// TwinCAT 3 PLC project PLC1
// ProgramVersion: 3.1.4022.7
// libraries:
//   Tc2_Standard, * (Beckhoff Automation GmbH)
//   Tc2_System, * (Beckhoff Automation GmbH)
//   Tc3_Module, * (Beckhoff Automation GmbH)
// project tree:
//   FBs/ FB_Publisher.TcPOU, FB_Subscriber.TcPOU
//   ITFs/ I_Publisher.TcIO, I_Subscriber.TcIO
//   / Param.TcGVL, PlcTask.TcTTO
//   POUs/ MAIN.TcPOU
// real-time tasks:
//   TASK PlcTask: cycle T#10ms, priority 20, ADS port 350

CONFIGURATION PLC1
    RESOURCE PLC ON TwinCAT3
        TASK PlcTask(INTERVAL := T#10ms, PRIORITY := 20);
        PROGRAM MAIN WITH PlcTask : MAIN;
    END_RESOURCE
END_CONFIGURATION

// ---- Param.TcGVL
{attribute 'qualified_only'}
VAR_GLOBAL CONSTANT
	MaxSubscribers : INT := 5;
END_VAR

// ---- ITFs/I_Publisher.TcIO
INTERFACE I_Publisher

METHOD AddSubscriber : BOOL
VAR_INPUT
	ipSubscriber : I_Subscriber;
END_VAR
END_METHOD

METHOD RemoveSubscriber : BOOL
VAR_INPUT
	ipSubscriber : I_Subscriber;
END_VAR
END_METHOD

END_INTERFACE

// ---- ITFs/I_Subscriber.TcIO
INTERFACE I_Subscriber

METHOD Update : BOOL
VAR_INPUT
	Value : LREAL;
END_VAR
END_METHOD

END_INTERFACE

// ---- POUs/MAIN.TcPOU
PROGRAM MAIN
VAR
	(*Design Pattern Blocks *)
	fbPublisher 	: FB_Publisher;
	fbSubscriber 	: ARRAY[1..Param.MaxSubscribers] OF FB_Subscriber;
	
	(* UI Values *)
	AddSub			: ARRAY[1..Param.MaxSubscribers] OF BOOL;
	DeleteSub		: ARRAY[1..Param.MaxSubscribers] OF BOOL;
	i				: INT;
END_VAR

fbPublisher();

FOR i := 1 TO Param.MaxSubscribers DO
	
	IF (AddSub[i]) THEN
		fbPublisher.AddSubscriber(fbSubscriber[i]);
		AddSub[i] := FALSE;
	END_IF

	IF (DeleteSub[i]) THEN
		fbPublisher.RemoveSubscriber(fbSubscriber[i]);
		DeleteSub[i] := FALSE;
	END_IF
	
END_FOR

END_PROGRAM

// ---- FBs/FB_Publisher.TcPOU
FUNCTION_BLOCK PUBLIC FB_Publisher IMPLEMENTS I_Publisher
VAR	
	fbDelay				: TON;
	fbDrand				: DRAND;
	_Value				: LREAL;
	aSubscribers		: ARRAY [1..Param.MaxSubscribers] OF I_Subscriber;
END_VAR

// creates every sec a random value and invoke the update method
fbDelay(IN := TRUE, PT := T#1S);
IF (fbDelay.Q) THEN	
	fbDelay(IN := FALSE);	
	fbDrand(SEED := 0);
	_Value := fbDrand.Num * 1234.5;
	NotifySubscribers();
END_IF

PROPERTY ActualValue : LREAL
GET
ActualValue := THIS^._Value;
END_GET
END_PROPERTY

METHOD PUBLIC AddSubscriber : BOOL
VAR_INPUT
	ipSubscriber	: I_Subscriber;
END_VAR
VAR
	nIndex					: INT := 0;
END_VAR
AddSubscriber := FALSE;
IF (ipSubscriber = 0) THEN
	RETURN;
END_IF

// is the observer already registered?
FOR nIndex := 1 TO Param.MaxSubscribers DO	
	IF (THIS^.aSubscribers[nIndex] = ipSubscriber) THEN
		RETURN;
	END_IF
END_FOR

// save the observer object into the array of observers and send the actual value
FOR nIndex := 1 TO Param.MaxSubscribers DO
	IF (THIS^.aSubscribers[nIndex] = 0) THEN
		THIS^.aSubscribers[nIndex] := ipSubscriber;
		THIS^.aSubscribers[nIndex].Update(THIS^._Value);
		AddSubscriber := TRUE;
		EXIT;					
	END_IF
END_FOR
END_METHOD

METHOD PRIVATE NotifySubscribers : BOOL
VAR	
	nIndex	: INT := 0;
END_VAR
FOR nIndex := 1 TO Param.MaxSubscribers DO
	IF (THIS^.aSubscribers[nIndex] <> 0) THEN
		THIS^.aSubscribers[nIndex].Update(THIS^.ActualValue);
	END_IF
END_FOR
END_METHOD

METHOD RemoveSubscriber : BOOL
VAR_INPUT
	ipSubscriber	: I_Subscriber;
END_VAR
VAR
	nIndex			: INT := 0;
END_VAR
RemoveSubscriber := FALSE;
IF (ipSubscriber = 0) THEN
	RETURN;
END_IF

FOR nIndex := 1 TO Param.MaxSubscribers DO
	IF (THIS^.aSubscribers[nIndex] = ipSubscriber) THEN
		THIS^.aSubscribers[nIndex] := 0;
		RemoveSubscriber := TRUE;	
	END_IF
END_FOR
END_METHOD

END_FUNCTION_BLOCK

// ---- FBs/FB_Subscriber.TcPOU
FUNCTION_BLOCK PUBLIC FB_Subscriber IMPLEMENTS I_Subscriber
VAR
	_Value				: LREAL;
END_VAR

PROPERTY ActualValue : LREAL
GET
ActualValue := THIS^._Value;
END_GET
END_PROPERTY

METHOD PUBLIC Update : BOOL
VAR_INPUT
	Value	: LREAL;
END_VAR
THIS^._Value := Value;
END_METHOD

END_FUNCTION_BLOCK
